PROGRAM VGC0
VAR
END_VAR

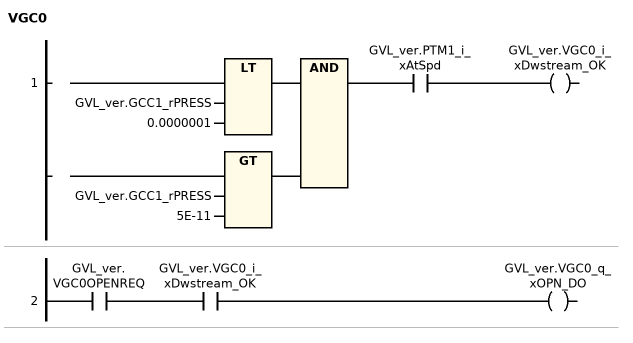
// NETWORK 1
GVL_ver.VGC0_i_xDwstream_OK := (GVL_ver.GCC1_rPRESS < 0.0000001 AND GVL_ver.GCC1_rPRESS > (5E-11)) AND GVL_ver.PTM1_i_xAtSpd;

// NETWORK 2
GVL_ver.VGC0_q_xOPN_DO := GVL_ver.VGC0OPENREQ AND GVL_ver.VGC0_i_xDwstream_OK;

END_PROGRAM

(* stored: Version 1.1.0.1, ProductVersion 3.1.4022.3
   POU VGC0: Id {5acfa6ce-8e0e-4447-bc74-7779d9f50280}, SpecialFunc None *)
